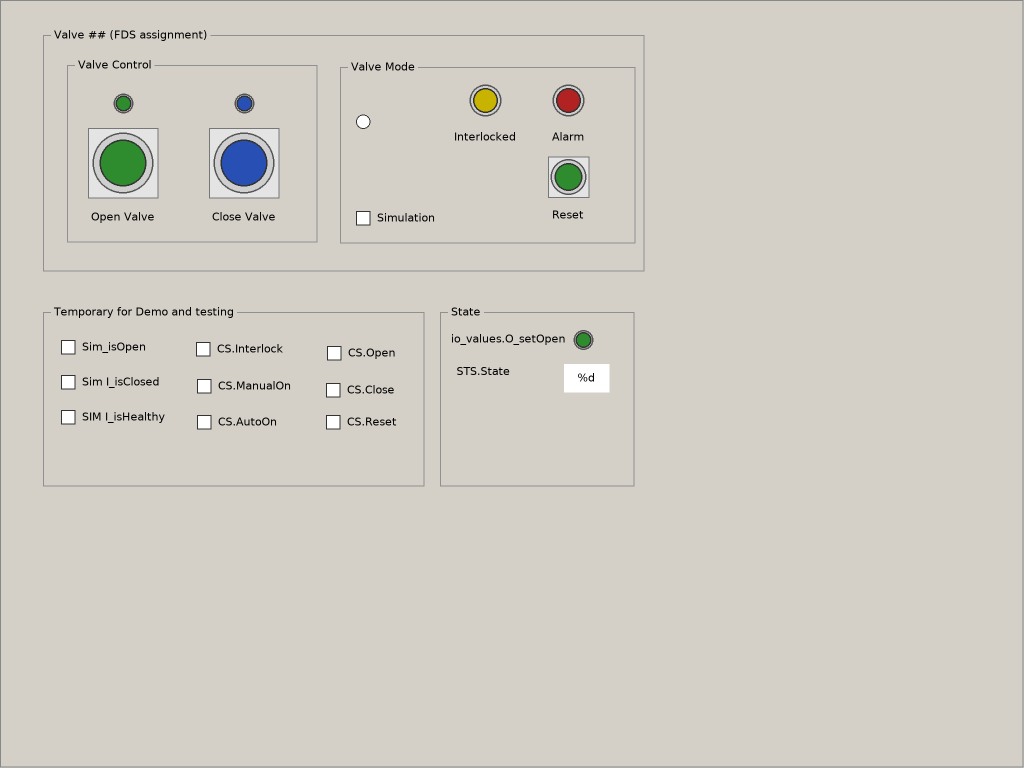
VISUALIZATION ValveHMI  // 1024x768
    GroupBox (43,27 601x244), "Valve ## (FDS assignment)"
        GroupBox (24,30 250x185), "Valve Control"
            PushSwitch (21,71 70x70), variable: GVL_VCM.valve01.Hmi.Open, behaviour: TOGGLE, style: Switch-PushSwitch-Green
            Lamp1 (45,35 23x23), variable: GVL_VCM.valve01.Sts.Open, style: Lamp-Lamp1-Green
            Label (14,145 84x30), "Open Valve"
            PushSwitch (142,71 70x70), variable: GVL_VCM.valve01.Hmi.Close, behaviour: TOGGLE, style: Switch-PushSwitch-Blue
            Label (135,145 84x30), "Close Valve"
            Lamp1 (166,35 23x23), variable: GVL_VCM.valve01.Sts.Closed, style: Lamp-Lamp1-Blue
        GroupBox (297,32 295x184), "Valve Mode"
            Lamp1 (210,22 37x39), variable: GVL_VCM.valve01.Alm.InAlarm, style: Lamp-Lamp1-Red
            Label (186,63 84x30), "Alarm"
            RadioButton (14,29 96x67), variable: GVL_VCM.valve01.Hmi.ModeValue, input disabled if: GVL_VCM.valve01.Hmi.DisableAutoManual
                Areas[0]: Text=Radiobutton
                Areas[1]: Text=Radiobutton
                p340057476: Manual
                p3123465237: Auto
                p2481256679: Interlock
            PushSwitch (208,93 41x50), variable: GVL_VCM.valve01.Hmi.Reset, behaviour: TOGGLE, style: Switch-PushSwitch-Green
            Label (186,141 84x30), "Reset"
            Label (103,63 84x30), "Interlocked"
            Lamp1 (127,22 37x39), variable: GVL_VCM.valve01.Sts.Interlock, style: Lamp-Lamp1-Yellow
            Checkbox (14,144 150x30), "Simulation", variable: GVL_VCM.valve01.Hmi.Simulation
    GroupBox (43,304 381x182), "Temporary for Demo and testing"
        Checkbox (16,28 133x30), "Sim_isOpen", variable: GVL_VCM.io_values.I_isOpen
        Checkbox (16,63 133x30), "Sim I_isClosed", variable: GVL_VCM.io_values.I_isClosed
        Checkbox (16,98 133x30), "SIM I_isHealthy", variable: GVL_VCM.io_values.I_isHealthy
        Checkbox (151,30 109x30), "CS.Interlock", variable: GVL_VCM.valve01.Cs.Interlock
        Checkbox (152,67 120x30), "CS.ManualOn", variable: GVL_VCM.valve01.Cs.ManualOn
        Checkbox (152,103 109x30), "CS.AutoOn", variable: GVL_VCM.valve01.Cs.AutoOn
        Checkbox (281,103 95x30), "CS.Reset", variable: GVL_VCM.valve01.Cs.Reset
        Checkbox (281,71 95x30), "CS.Close", variable: GVL_VCM.valve01.Cs.Close
        Checkbox (282,34 93x30), "CS.Open", variable: GVL_VCM.valve01.Cs.Open
    GroupBox (440,304 194x182), "State"
        Lamp1 (132,24 23x24), variable: GVL_VCM.io_values.O_setOpen, style: Lamp-Lamp1-Green
        Label (2,20 133x30), "io_values.O_setOpen"
        Label (74,91 53x30)
        Label (9,54 69x27), "STS.State"
        Textfield (123,59 47x30), "%d", text variable: GVL_VCM.valve01.Sts.State
END_VISUALIZATION

(* stored: Version 1.1.0.1, ProductVersion 3.1.4024.12
   Visu ValveHMI: Id {4057c5f4-4926-4faa-9281-d4bfa35f02eb} *)
